// TwinCAT 3 PLC project PLC
// ProgramVersion: 3.1.4023.0
// libraries:
//   CmpBitmapPool, * (System)
//   Tc2_Standard, * (Beckhoff Automation GmbH)
//   Tc2_System, * (Beckhoff Automation GmbH)
//   Tc3_Module, * (Beckhoff Automation GmbH)
// project tree:
//   / GlobalTextList.TcGTLO, PlcTask.TcTTO, VISU_TASK.TcTTO
//   GVLs/ GVL_IO.TcGVL
//   POUs/ FB_Scale.TcPOU, MAIN.TcPOU, PRG_IO_Scaling.TcPOU
//   VISUs/ Analog_Outputs.TcVIS, Digital_Inputs.TcVIS, Analog_Inputs.TcVIS, Digital_Outputs.TcVIS, ImagePool.TcIPO (not stored), Visualization.TcVIS, VisualizationManager.TcVMO (not stored)
// real-time tasks:
//   TASK PlcTask: cycle T#10ms, priority 20, ADS port 350
//   TASK VISU_TASK: cycle T#200000us, priority 30, ADS port 351
// I/O:
//   DEVICE Device 1 (EtherCAT), AmsNetId 5.47.207.56.2.1
//     Term 1 (EK1100) [EK1100 EtherCAT Coupler (2A E-Bus)]
//       Term 2 (EL1008) [EL1008 8Ch. Dig. Input 24V, 3ms]
//       Term 3 (EL3058) [EL3058 8Ch. Ana. Input 4-20mA]
//       Term 4 (EL4028) [EL4028 8Ch. Ana. Output 4-20mA, 12bit]
//       Term 5 (EL2809) [EL2809 16Ch. Dig. Output 24V, 0.5A]
//       Term 6 (EL9011) [EL9011 End Terminal]
//   DEVICE Device 2 (EtherCAT Automation Protocol), AmsNetId 5.47.207.56.3.1
// variable links:
//   PLC/PLC Instance <-> Device 1 (EtherCAT)/Term 1 (EK1100)/Term 2 (EL1008)
//     PlcTask Inputs/GVL_IO.DI{1..8} <-> Channel {1..8}/Input  (8 links)
//   PLC/PLC Instance <-> Device 1 (EtherCAT)/Term 1 (EK1100)/Term 3 (EL3058)
//     PlcTask Inputs/GVL_IO.AI{1..8} <-> AI Standard Channel {1..8}/Value  (8 links)
//   PLC/PLC Instance <-> Device 1 (EtherCAT)/Term 1 (EK1100)/Term 4 (EL4028)
//     PlcTask Outputs/GVL_IO.AO{1..8} <-> AO Outputs Channel {1..8}/Analog output  (8 links)
//   PLC/PLC Instance <-> Device 1 (EtherCAT)/Term 1 (EK1100)/Term 5 (EL2809)
//     PlcTask Outputs/GVL_IO.DO{1..16} <-> Channel {1..16}/Output  (16 links)
//   PLC/PLC Instance <-> Device 2 (EtherCAT Automation Protocol)
//     PlcTask Inputs/GVL_IO.sync_master_dev2 <-> Inputs/DevState

CONFIGURATION PLC
    RESOURCE PLC ON TwinCAT3
        TASK PlcTask(INTERVAL := T#10ms, PRIORITY := 20);
        TASK VISU_TASK(INTERVAL := T#200000us, PRIORITY := 30);
        PROGRAM MAIN WITH PlcTask : MAIN;
        PROGRAM PRG_IO_Scaling WITH PlcTask : PRG_IO_Scaling;
        PROGRAM VisuElems_Visu_Prg WITH VISU_TASK : VisuElems.Visu_Prg;
    END_RESOURCE
END_CONFIGURATION

// ---- GVLs/GVL_IO.TcGVL
{attribute 'qualified_only'}
VAR_GLOBAL
	sync_master_dev2 AT %I*: UINT;
	AI1 AT %I*: INT;	
	AI2 AT %I*: INT;
	AI3 AT %I*: INT;
	AI4 AT %I*: INT;
	AI5 AT %I*: INT;
	AI6 AT %I*: INT;
	AI7 AT %I*: INT;
	AI8 AT %I*: INT;
	
	AO1 AT %Q*: INT;
	AO2 AT %Q*: INT;
	AO3 AT %Q*: INT;
	AO4 AT %Q*: INT;
	AO5 AT %Q*: INT;
	AO6 AT %Q*: INT;
	AO7 AT %Q*: INT;
	AO8 AT %Q*: INT;
	
	DI1 AT %I*: BOOL;
	DI2 AT %I*: BOOL;
	DI3 AT %I*: BOOL;
	DI4 AT %I*: BOOL;
	DI5 AT %I*: BOOL;
	DI6 AT %I*: BOOL;
	DI7 AT %I*: BOOL;
	DI8 AT %I*: BOOL;
	
	DO1 AT %Q*: BOOL;
	DO2 AT %Q*: BOOL;
	DO3 AT %Q*: BOOL;
	DO4 AT %Q*: BOOL;
	DO5 AT %Q*: BOOL;
	DO6 AT %Q*: BOOL;
	DO7 AT %Q*: BOOL;
	DO8 AT %Q*: BOOL;
	DO9 AT %Q*: BOOL;
	DO10 AT %Q*: BOOL;
	DO11 AT %Q*: BOOL;
	DO12 AT %Q*: BOOL;
	DO13 AT %Q*: BOOL;
	DO14 AT %Q*: BOOL;
	DO15 AT %Q*: BOOL;
	DO16 AT %Q*: BOOL;
	AI1_ENG: REAL;
	AI2_ENG: REAL;
	AI3_ENG: REAL;
	AI4_ENG: REAL;
	AI5_ENG: REAL;
	AI6_ENG: REAL;
	AI7_ENG: REAL;
	AI8_ENG: REAL;
	AO1_SET: REAL;
	AO2_SET: REAL;
	AO3_SET: REAL;
	AO4_SET: REAL;
	AO5_SET: REAL;
	AO6_SET: REAL;
	AO7_SET: REAL;
	AO8_SET: REAL;
	
END_VAR

// ---- POUs/MAIN.TcPOU
PROGRAM MAIN

END_PROGRAM

// ---- POUs/PRG_IO_Scaling.TcPOU
PROGRAM PRG_IO_Scaling
VAR
	AI1: FB_Scale;
	AI2: FB_Scale;
	AI3: FB_Scale;
	AI4: FB_Scale;
	AI5: FB_Scale;
	AI6: FB_Scale;
	AI7: FB_Scale;
	AI8: FB_Scale;
	AO1: FB_Scale;
	AO2: FB_Scale;
	AO3: FB_Scale;
	AO4: FB_Scale;
	AO5: FB_Scale;
	AO6: FB_Scale;
	AO7: FB_Scale;
	AO8: FB_Scale;
END_VAR

AI1(X_MIN := 0, X_MAX := 4096, Y_MIN := 4, Y_MAX := 20, IN_VALUE := GVL_IO.AI1); // FB_Scale
GVL_IO.AI1_ENG := AI1.OUT_VALUE;
AI5(X_MIN := 0, X_MAX := 4096, Y_MIN := 4, Y_MAX := 20, IN_VALUE := GVL_IO.AI5); // FB_Scale
GVL_IO.AI5_ENG := AI5.OUT_VALUE;
AI2(X_MIN := 0, X_MAX := 4096, Y_MIN := 4, Y_MAX := 20, IN_VALUE := GVL_IO.AI2); // FB_Scale
GVL_IO.AI2_ENG := AI2.OUT_VALUE;
AI6(X_MIN := 0, X_MAX := 4096, Y_MIN := 4, Y_MAX := 20, IN_VALUE := GVL_IO.AI6); // FB_Scale
GVL_IO.AI6_ENG := AI6.OUT_VALUE;
AI3(X_MIN := 0, X_MAX := 4096, Y_MIN := 4, Y_MAX := 20, IN_VALUE := GVL_IO.AI3); // FB_Scale
GVL_IO.AI3_ENG := AI3.OUT_VALUE;
AI7(X_MIN := 0, X_MAX := 4096, Y_MIN := 4, Y_MAX := 20, IN_VALUE := GVL_IO.AI7); // FB_Scale
GVL_IO.AI7_ENG := AI7.OUT_VALUE;
AI4(X_MIN := 0, X_MAX := 4096, Y_MIN := 4, Y_MAX := 20, IN_VALUE := GVL_IO.AI4); // FB_Scale
GVL_IO.AI4_ENG := AI4.OUT_VALUE;
AI8(X_MIN := 0, X_MAX := 4096, Y_MIN := 4, Y_MAX := 20, IN_VALUE := GVL_IO.AI8); // FB_Scale
GVL_IO.AI8_ENG := AI8.OUT_VALUE;
AO1(X_MIN := 4, X_MAX := 20, Y_MIN := 0, Y_MAX := 4096, IN_VALUE := GVL_IO.AO1_SET); // FB_Scale
GVL_IO.AO1 := REAL_TO_INT(AO1.OUT_VALUE);
AO5(X_MIN := 4, X_MAX := 20, Y_MIN := 0, Y_MAX := 4096, IN_VALUE := GVL_IO.AO5_SET); // FB_Scale
GVL_IO.AO5 := REAL_TO_INT(AO5.OUT_VALUE);
AO2(X_MIN := 4, X_MAX := 20, Y_MIN := 0, Y_MAX := 4096, IN_VALUE := GVL_IO.AO2_SET); // FB_Scale
GVL_IO.AO2 := REAL_TO_INT(AO2.OUT_VALUE);
AO6(X_MIN := 4, X_MAX := 20, Y_MIN := 0, Y_MAX := 4096, IN_VALUE := GVL_IO.AO6_SET); // FB_Scale
GVL_IO.AO6 := REAL_TO_INT(AO6.OUT_VALUE);
AO3(X_MIN := 4, X_MAX := 20, Y_MIN := 0, Y_MAX := 4096, IN_VALUE := GVL_IO.AO3_SET); // FB_Scale
GVL_IO.AO3 := REAL_TO_INT(AO3.OUT_VALUE);
AO7(X_MIN := 4, X_MAX := 20, Y_MIN := 0, Y_MAX := 4096, IN_VALUE := GVL_IO.AO7_SET); // FB_Scale
GVL_IO.AO7 := REAL_TO_INT(AO7.OUT_VALUE);
AO4(X_MIN := 4, X_MAX := 20, Y_MIN := 0, Y_MAX := 4096, IN_VALUE := GVL_IO.AO4_SET); // FB_Scale
GVL_IO.AO4 := REAL_TO_INT(AO4.OUT_VALUE);
AO8(X_MIN := 4, X_MAX := 20, Y_MIN := 0, Y_MAX := 4096, IN_VALUE := GVL_IO.AO8_SET); // FB_Scale
GVL_IO.AO8 := REAL_TO_INT(AO8.OUT_VALUE);

END_PROGRAM

// ---- POUs/FB_Scale.TcPOU
FUNCTION_BLOCK FB_Scale
VAR_INPUT
	X_MIN: REAL;
	X_MAX: REAL;
	Y_MIN: REAL;
	Y_MAX: REAL;
	IN_VALUE: REAL;
END_VAR
VAR_OUTPUT
	OUT_VALUE: REAL;
END_VAR
VAR
	a: REAL;
END_VAR

a := (Y_MAX - Y_MIN) / (X_MAX - X_MIN);
OUT_VALUE := a*(IN_VALUE-X_MIN) + Y_MIN;

END_FUNCTION_BLOCK

// ---- GlobalTextList.TcGTLO
TEXTLIST GlobalTextList
  447 = 'AI'
  381 = 'AI1'
  740 = 'AI2'
  233 = 'AI3'
  765 = 'AI4'
  985 = 'AI5'
  641 = 'AI6'
  453 = 'AI7'
  289 = 'AI8'
  431 = 'AO'
  134 = 'AO1'
  640 = 'AO2'
  846 = 'AO3'
  369 = 'AO4'
  935 = 'AO5'
  800 = 'AO6'
  857 = 'AO7'
  328 = 'AO8'
  20 = 'DI'
  154 = 'DI1'
  906 = 'DI10'
  53 = 'DI11'
  472 = 'DI12'
  894 = 'DI13'
  56 = 'DI14'
  116 = 'DI15'
  357 = 'DI16'
  557 = 'DI2'
  774 = 'DI3'
  408 = 'DI4'
  28 = 'DI5'
  252 = 'DI6'
  172 = 'DI7'
  891 = 'DI8'
  863 = 'DI9'
  533 = 'DO'
  881 = 'DO1'
  623 = 'DO10'
  773 = 'DO11'
  200 = 'DO12'
  598 = 'DO13'
  494 = 'DO14'
  251 = 'DO15'
  119 = 'DO16'
  105 = 'DO2'
  179 = 'DO3'
  9 = 'DO4'
  929 = 'DO5'
  45 = 'DO6'
  732 = 'DO7'
  366 = 'DO8'
  301 = 'DO9'
  764 = 'Przycisk'
END_TEXTLIST

// ---- VISUs/Analog_Outputs.TcVIS
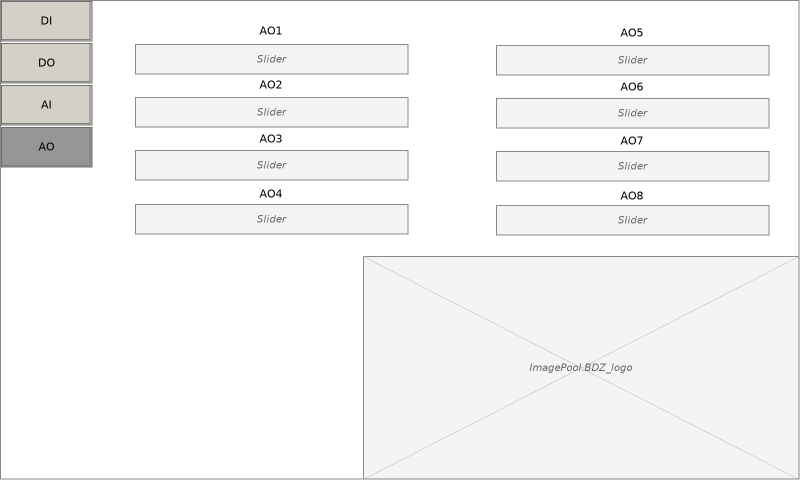
VISUALIZATION Analog_Outputs  // 800x480
    Slider (135,44 273x30), variable: GVL_IO.AO1_SET, scale 4..20
    Slider (135,97 273x30), variable: GVL_IO.AO2_SET, scale 4..20
    Slider (135,150 273x30), variable: GVL_IO.AO3_SET, scale 4..20
    Slider (135,204 273x30), variable: GVL_IO.AO4_SET, scale 4..20
    Slider (496,45 273x30), variable: GVL_IO.AO5_SET, scale 4..20
    Slider (496,98 273x30), variable: GVL_IO.AO6_SET, scale 4..20
    Slider (496,151 273x30), variable: GVL_IO.AO7_SET, scale 4..20
    Slider (496,205 273x30), variable: GVL_IO.AO8_SET, scale 4..20
    Label (196,16 150x30), "AO1"
    Label (196,70 150x30), "AO2"
    Label (196,124 150x30), "AO3"
    Label (196,179 150x30), "AO4"
    Label (557,18 150x30), "AO5"
    Label (557,72 150x30), "AO6"
    Label (557,126 150x30), "AO7"
    Label (557,181 150x30), "AO8"
    Button (1,127 91x40), "AO"
        OnMouseUp: change screen: Analog_Outputs
    Button (1,1 91x40), "DI"
        OnMouseUp: change screen: Digital_Inputs
    Button (1,43 91x40), "DO"
        OnMouseDown: change screen: Digital_Outputs
        OnMouseUp: change screen: Digital_Outputs
    Button (1,85 91x40), "AI"
        OnMouseUp: change screen: Analog_Inputs
    Image (363,256 436x223), image: ImagePool.BDZ_logo
END_VISUALIZATION

// ---- VISUs/Digital_Inputs.TcVIS
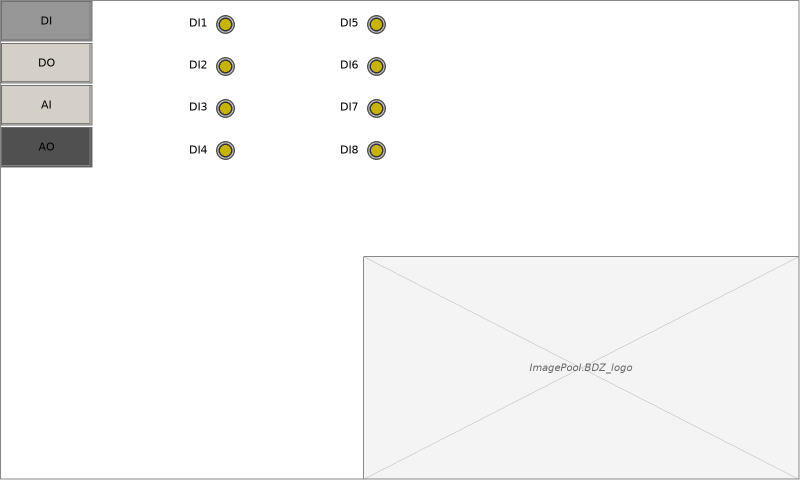
VISUALIZATION Digital_Inputs  // 800x480
    Button (1,127 91x40), "AO"
        OnMouseUp: change screen: Analog_Outputs
    Button (1,1 91x40), "DI"
        OnMouseUp: change screen: Digital_Inputs
    Button (1,43 91x40), "DO"
        OnMouseDown: change screen: Digital_Outputs
        OnMouseUp: change screen: Digital_Outputs
    Button (1,85 91x40), "AI"
        OnMouseUp: change screen: Analog_Inputs
    Lamp1 (215,14 21x21), variable: GVL_IO.DI1, style: Lamp-Lamp1-Yellow
    Lamp1 (215,56 21x21), variable: GVL_IO.DI2, style: Lamp-Lamp1-Yellow
    Lamp1 (215,98 21x21), variable: GVL_IO.DI3, style: Lamp-Lamp1-Yellow
    Lamp1 (215,140 21x21), variable: GVL_IO.DI4, style: Lamp-Lamp1-Yellow
    Label (179,8 39x30), "DI1"
    Label (179,50 39x30), "DI2"
    Label (179,92 39x30), "DI3"
    Label (179,135 39x30), "DI4"
    Lamp1 (366,14 21x21), variable: GVL_IO.DI5, style: Lamp-Lamp1-Yellow
    Lamp1 (366,56 21x21), variable: GVL_IO.DI6, style: Lamp-Lamp1-Yellow
    Lamp1 (366,98 21x21), variable: GVL_IO.DI7, style: Lamp-Lamp1-Yellow
    Lamp1 (366,140 21x21), variable: GVL_IO.DI8, style: Lamp-Lamp1-Yellow
    Label (330,8 39x30), "DI5"
    Label (330,50 39x30), "DI6"
    Label (330,92 39x30), "DI7"
    Label (330,135 39x30), "DI8"
    Image (363,256 436x223), image: ImagePool.BDZ_logo
END_VISUALIZATION

// ---- VISUs/Analog_Inputs.TcVIS
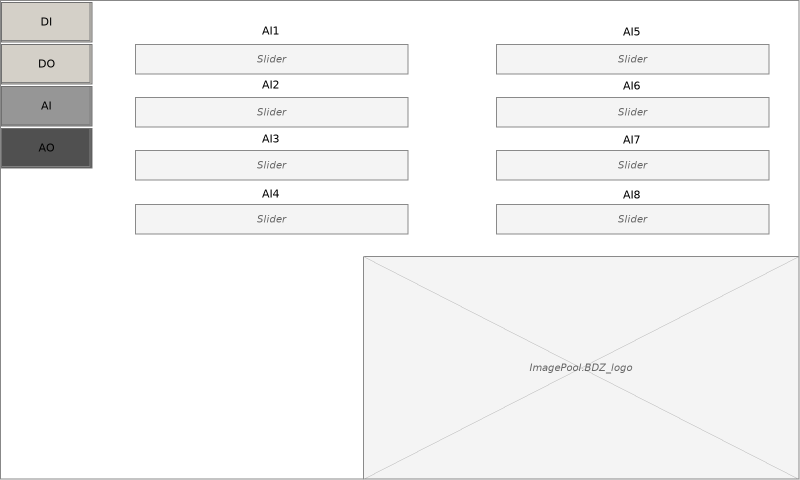
VISUALIZATION Analog_Inputs  // 800x480
    Slider (135,44 273x30), variable: GVL_IO.AI1_ENG, scale 4..20
    Slider (135,97 273x30), variable: GVL_IO.AI2_ENG, scale 4..20
    Slider (135,150 273x30), variable: GVL_IO.AI3_ENG, scale 4..20
    Slider (135,204 273x30), variable: GVL_IO.AI4_ENG, scale 4..20
    Slider (496,44 273x30), variable: GVL_IO.AI5_ENG, scale 4..20
    Slider (496,97 273x30), variable: GVL_IO.AI6_ENG, scale 4..20
    Slider (496,150 273x30), variable: GVL_IO.AI7_ENG, scale 4..20
    Slider (496,204 273x30), variable: GVL_IO.AI8_ENG, scale 4..20
    Label (196,16 150x30), "AI1"
    Label (196,70 150x30), "AI2"
    Label (196,124 150x30), "AI3"
    Label (196,179 150x30), "AI4"
    Label (557,17 150x30), "AI5"
    Label (557,71 150x30), "AI6"
    Label (557,125 150x30), "AI7"
    Label (557,180 150x30), "AI8"
    Button (1,128 91x40), "AO"
        OnMouseUp: change screen: Analog_Outputs
    Button (1,2 91x40), "DI"
        OnMouseUp: change screen: Digital_Inputs
    Button (1,44 91x40), "DO"
        OnMouseDown: change screen: Digital_Outputs
        OnMouseUp: change screen: Digital_Outputs
    Button (1,86 91x40), "AI"
        OnMouseUp: change screen: Analog_Inputs
    Image (363,256 436x223), image: ImagePool.BDZ_logo
END_VISUALIZATION

// ---- VISUs/Digital_Outputs.TcVIS
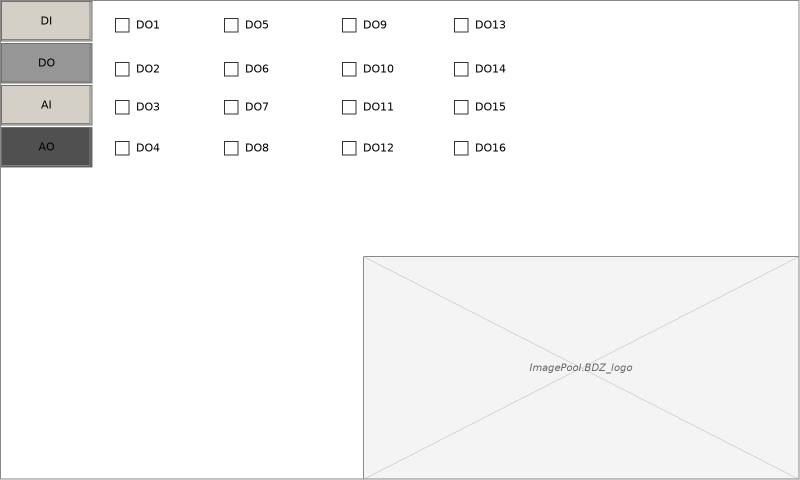
VISUALIZATION Digital_Outputs  // 800x480
    Button (1,127 91x40), "AO"
        OnMouseUp: change screen: Analog_Outputs
    Button (1,1 91x40), "DI"
        OnMouseUp: change screen: Digital_Inputs
    Button (1,43 91x40), "DO"
        OnMouseDown: change screen: Digital_Outputs
        OnMouseUp: change screen: Digital_Outputs
    Button (1,85 91x40), "AI"
        OnMouseUp: change screen: Analog_Inputs
    Checkbox (113,10 62x30), "DO1", variable: GVL_IO.DO1
    Checkbox (113,54 62x30), "DO2", variable: GVL_IO.DO2
    Checkbox (113,92 62x30), "DO3", variable: GVL_IO.DO3
    Checkbox (113,133 62x30), "DO4", variable: GVL_IO.DO4
    Checkbox (222,10 62x30), "DO5", variable: GVL_IO.DO5
    Checkbox (222,54 62x30), "DO6", variable: GVL_IO.DO6
    Checkbox (222,92 62x30), "DO7", variable: GVL_IO.DO7
    Checkbox (222,133 62x30), "DO8", variable: GVL_IO.DO8
    Checkbox (340,10 62x30), "DO9", variable: GVL_IO.DO9
    Checkbox (340,54 74x30), "DO10", variable: GVL_IO.DO10
    Checkbox (340,92 71x30), "DO11", variable: GVL_IO.DO11
    Checkbox (340,133 72x30), "DO12", variable: GVL_IO.DO12
    Checkbox (452,10 69x30), "DO13", variable: GVL_IO.DO13
    Checkbox (452,54 80x30), "DO14", variable: GVL_IO.DO14
    Checkbox (452,92 72x30), "DO15", variable: GVL_IO.DO15
    Checkbox (452,133 77x30), "DO16", variable: GVL_IO.DO16
    Image (363,256 436x223), image: ImagePool.BDZ_logo
END_VISUALIZATION

// ---- VISUs/Visualization.TcVIS
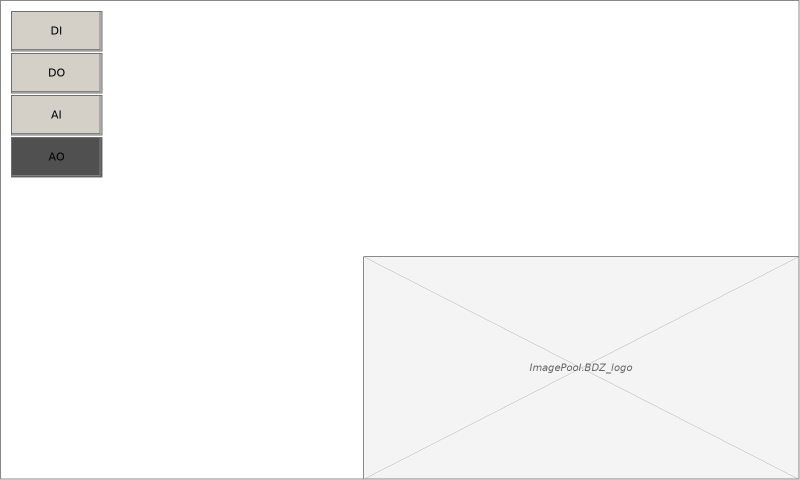
VISUALIZATION Visualization  // 800x480
    Image (363,256 436x223), image: ImagePool.BDZ_logo
    Button (11,11 91x40), "DI"
        OnMouseUp: change screen: Digital_Inputs
    Button (11,53 91x40), "DO"
        OnMouseDown: change screen: Digital_Outputs
        OnMouseUp: change screen: Digital_Outputs
    Button (11,95 91x40), "AI"
        OnMouseUp: change screen: Analog_Inputs
    Button (11,137 91x40), "AO"
        OnMouseUp: change screen: Analog_Outputs
END_VISUALIZATION
